FUNCTION_BLOCK Necessidade_2_Equipamentos (* Composite Function Block Type *)
  (* Standard: 61499-2 *)
  (* Version 0.0, 25/02/2026, template *)
  PACKAGE Hidryco.HidrycoLib;
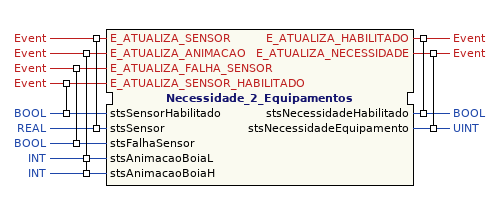
  EVENT_INPUT
    E_ATUALIZA_SENSOR WITH stsSensor;
    E_ATUALIZA_ANIMACAO WITH stsAnimacaoBoiaL, stsAnimacaoBoiaH;
    E_ATUALIZA_FALHA_SENSOR WITH stsFalhaSensor;
    E_ATUALIZA_SENSOR_HABILITADO WITH stsSensorHabilitado;
  END_EVENT
  EVENT_OUTPUT
    E_ATUALIZA_HABILITADO WITH stsNecessidadeHabilitado;
    E_ATUALIZA_NECESSIDADE WITH stsNecessidadeEquipamento;
  END_EVENT
  VAR_INPUT
    stsSensorHabilitado : BOOL;
    stsSensor : REAL;
    stsFalhaSensor : BOOL;
    stsAnimacaoBoiaL : INT;
    stsAnimacaoBoiaH : INT;
  END_VAR
  VAR_OUTPUT
    stsNecessidadeHabilitado : BOOL;
    stsNecessidadeEquipamento : UINT;
  END_VAR
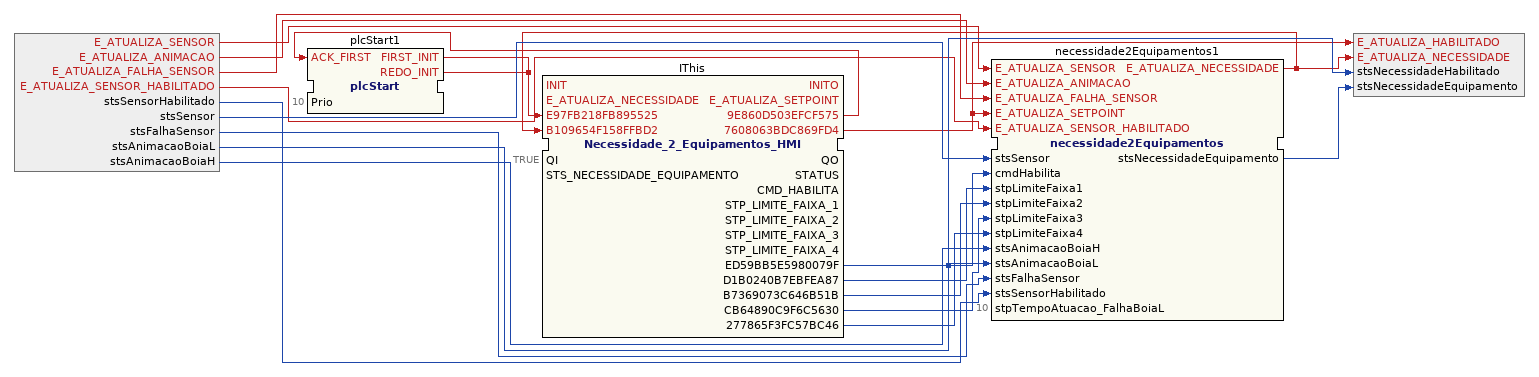
  FBS
    IThis : Necessidade_2_Equipamentos_HMI(QI := TRUE);
    plcStart1 : plcStart(Prio := 10);
    necessidade2Equipamentos1 : necessidade2Equipamentos(stpTempoAtuacao_FalhaBoiaL := 10);
  END_FBS
  EVENT_CONNECTIONS
    E_ATUALIZA_SENSOR TO necessidade2Equipamentos1.E_ATUALIZA_SENSOR;
    E_ATUALIZA_ANIMACAO TO necessidade2Equipamentos1.E_ATUALIZA_ANIMACAO;
    E_ATUALIZA_FALHA_SENSOR TO necessidade2Equipamentos1.E_ATUALIZA_FALHA_SENSOR;
    plcStart1.FIRST_INIT TO IThis.E97FB218FB895525;
    plcStart1.REDO_INIT TO IThis.E97FB218FB895525;
    necessidade2Equipamentos1.E_ATUALIZA_NECESSIDADE TO IThis.B109654F158FFBD2;
    IThis.9E860D503EFCF575 TO plcStart1.ACK_FIRST;
    IThis.7608063BDC869FD4 TO necessidade2Equipamentos1.E_ATUALIZA_SETPOINT;
    necessidade2Equipamentos1.E_ATUALIZA_NECESSIDADE TO E_ATUALIZA_NECESSIDADE;
    IThis.7608063BDC869FD4 TO E_ATUALIZA_HABILITADO;
    E_ATUALIZA_SENSOR_HABILITADO TO necessidade2Equipamentos1.E_ATUALIZA_SENSOR_HABILITADO;
  END_CONNECTIONS
  DATA_CONNECTIONS
    stsSensor TO necessidade2Equipamentos1.stsSensor;
    necessidade2Equipamentos1.stsNecessidadeEquipamento TO stsNecessidadeEquipamento;
    IThis.ED59BB5E5980079F TO necessidade2Equipamentos1.cmdHabilita;
    IThis.D1B0240B7EBFEA87 TO necessidade2Equipamentos1.stpLimiteFaixa1;
    IThis.B7369073C646B51B TO necessidade2Equipamentos1.stpLimiteFaixa2;
    IThis.CB64890C9F6C5630 TO necessidade2Equipamentos1.stpLimiteFaixa3;
    IThis.277865F3FC57BC46 TO necessidade2Equipamentos1.stpLimiteFaixa4;
    stsAnimacaoBoiaH TO necessidade2Equipamentos1.stsAnimacaoBoiaH;
    stsAnimacaoBoiaL TO necessidade2Equipamentos1.stsAnimacaoBoiaL;
    stsFalhaSensor TO necessidade2Equipamentos1.stsFalhaSensor;
    IThis.ED59BB5E5980079F TO stsNecessidadeHabilitado;
    stsSensorHabilitado TO necessidade2Equipamentos1.stsSensorHabilitado;
  END_CONNECTIONS
END_FUNCTION_BLOCK
